// TIA Portal V20 export
DATA_BLOCK "instFB_PatternAutoGen"   // DB25
VERSION : 1.1
// stored: InstanceOfName FB_PatternAutoGen, InstanceOfType FB
"FB_PatternAutoGen"
   // VAR
   //    statCyclePalletIdx : Int;   // V3.0 (2026-05-23): which pallet's cycle is currently in flight. Snapshotted from i16_ActivePalletIdx at the rising edge of GDB_PalletizingCmd.bo_InitPallet. Used by LatchPalletFull region to correctly attribute bo_PalletDone to the pallet whose cycle is completing -- even if operator has swapped activeIdx mid-cycle (or released both flags). 0 = no cycle in progress.
   //    statInitPallet_prev : Bool;   // V3.0: previous-scan value of GDB_PalletizingCmd.bo_InitPallet for rising-edge detection in TrackCycleStart region.
   // END_VAR
BEGIN
END_DATA_BLOCK
